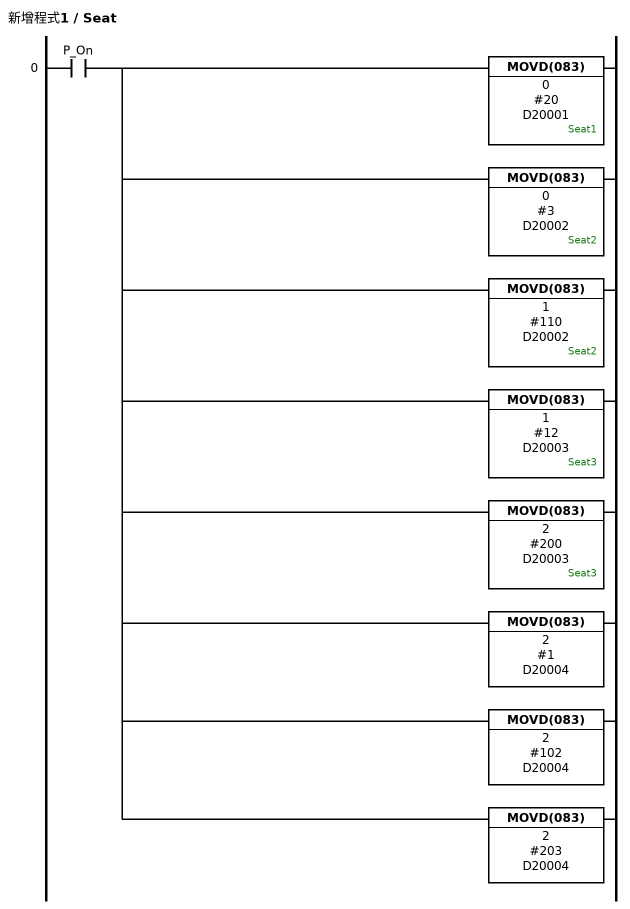
; [picture p24: 新增程式1 / Seat, rungs 0-0]
; rung 0
LD P_On
MOVD(083) 0 #20 D20001  ; Seat1
MOVD(083) 0 #3 D20002  ; Seat2
MOVD(083) 1 #110 D20002  ; Seat2
MOVD(083) 1 #12 D20003  ; Seat3
MOVD(083) 2 #200 D20003  ; Seat3
MOVD(083) 2 #1 D20004
MOVD(083) 2 #102 D20004
MOVD(083) 2 #203 D20004

### Section 純水補

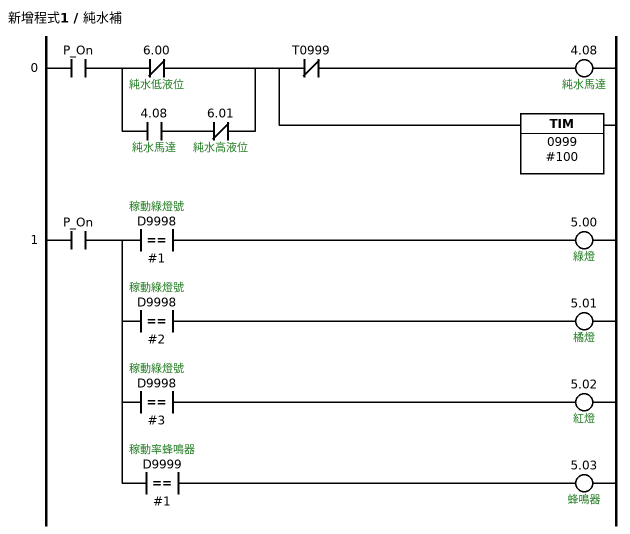
; rung 0
LD P_On
LDNOT 6.00  ; 純水低液位
LD 4.08  ; 純水馬達
ANDNOT 6.01  ; 純水高液位
ORLD
ANDLD
OUT TR0
ANDNOT T0999
OUT 4.08  ; 純水馬達
LD TR0
TIM 0999 #100
; rung 1
LD P_On
OUT TR0
AND=(300) D9998 #1  ; 稼動綠燈號
OUT 5.00  ; 綠燈
LD TR0
AND=(300) D9998 #2  ; 稼動綠燈號
OUT 5.01  ; 橘燈
LD TR0
AND=(300) D9998 #3  ; 稼動綠燈號
OUT 5.02  ; 紅燈
LD TR0
AND=(300) D9999 #1  ; 稼動率蜂鳴器
OUT 5.03  ; 蜂鳴器

### Section END
; rung 0
END(001)